FUNCTION_BLOCK MY_X2Y2_J (* Compute X^2-Y^2 in ST *)
  (* Standard: 61499-1 *)
  (* Version 0.0, 2002-09-24, JHC, Rockwell Automation, Derived from FB_X2Y2_J. *)
  (* Compiler header: package fb.rt.student; *)
  (* Compiler Java IBM Jikes 1.0.6 *)
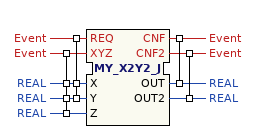
  EVENT_INPUT
    REQ WITH Y, X;
    XYZ WITH Y, X, Z;
  END_EVENT
  EVENT_OUTPUT
    CNF WITH OUT;
    CNF2 WITH OUT2;
  END_EVENT
  VAR_INPUT
    X : REAL;
    Y : REAL;
    Z : REAL;
  END_VAR
  VAR_OUTPUT
    OUT : REAL;
    OUT2 : REAL;
  END_VAR
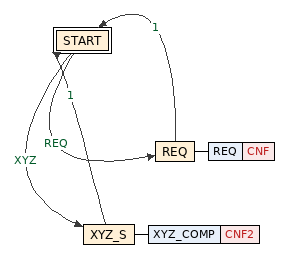
  EC_STATES
    START;
    REQ : REQ -> CNF;
    XYZ_S : XYZ_COMP -> CNF2;
  END_STATES
  EC_TRANSITIONS
    START TO REQ := REQ;
    REQ TO START := 1;
    START TO XYZ_S := XYZ;
    XYZ_S TO START := 1;
  END_TRANSITIONS
  ALGORITHM REQ IN Java:
OUT.value = X.value*X.value+Y.value*Y.value;
  END_ALGORITHM
  ALGORITHM XYZ_COMP IN Java:
OUT2.value = X.value + Y.value + Z.value;
System.out.println("This is in algorithm XYZ");
  END_ALGORITHM
END_FUNCTION_BLOCK
